// TIA Portal V19 export
VAR_GLOBAL   // PLC tag table "A03_303"
   A0303_Spalla_Ax_Testa_Posizionamento_Ls_Minimo AT %I355.7 : Bool;   // 2262SQ1
   A0303_Spalla_Ax_Testa_Posizionamento_Ls_Massimo AT %I356.0 : Bool;   // 2262SQ2
   A0303_Spintore_Testa_Verticale_Ls_Rest AT %I356.1 : Bool;   // 2270SQ1
   A0303_Spintore_Testa_Verticale_Ls_Work AT %I356.2 : Bool;   // 2270SQ2
   A0303_Spintore_Testa_Orizzontale_Ls_Rest AT %I356.3 : Bool;   // 2270SQ3
   A0303_Spintore_Testa_Orizzontale_Ls_Work AT %I356.4 : Bool;   // 2270SQ4
   A0303_Spintore_Testa_Verticale_V_Rest AT %Q362.2 : Bool;   // 2270YV1
   A0303_Spintore_Testa_Verticale_V_Work AT %Q362.3 : Bool;   // 2270YV2
   A0303_Spintore_Testa_Orizzontale_V_Rest AT %Q362.4 : Bool;   // 2270YV3
   A0303_Spintore_Testa_Orizzontale_V_Work AT %Q362.5 : Bool;   // 2270YV4
   A0303_ControlloPezzo_Testa_Phc_InPosizione AT %I356.5 : Bool;   // 2271BF1
   A0303_ControlloPezzo_Testa_Phc_MassimaPosizione AT %I356.6 : Bool;   // 2271BF2
   A0303_SostegnoStrato_Testa_Verticale_Ls_Alto AT %I356.7 : Bool;   // 2274SQ1
   A0303_SostegnoStrato_Testa_Verticale_Ls_Basso AT %I357.0 : Bool;   // 2274SQ2
   A0303_SostegnoStrato_Testa_Verticale_V_Alto AT %Q362.6 : Bool;   // 2274YV1
   A0303_SostegnoStrato_Testa_Verticale_V_Basso AT %Q362.7 : Bool;   // 2274YV2
   A0303_Spalla_Ax_Coda_Posizionamento_Ls_Minimo AT %I305.7 : Bool;   // 2282SQ1
   A0303_Spalla_Ax_Coda_Posizionamento_Ls_Massimo AT %I306.0 : Bool;   // 2282SQ2
   A0303_Spintore_Coda_Verticale_Ls_Rest AT %I306.1 : Bool;   // 2300SQ1
   A0303_Spintore_Coda_Verticale_Ls_Work AT %I306.2 : Bool;   // 2300SQ2
   A0303_Spintore_Coda_Orizzontale_Ls_Rest AT %I306.3 : Bool;   // 2300SQ3
   A0303_Spintore_Coda_Orizzontale_Ls_Work AT %I306.4 : Bool;   // 2300SQ4
   A0303_Spintore_Coda_Verticale_V_Rest AT %Q311.6 : Bool;   // 2300YV1
   A0303_Spintore_Coda_Verticale_V_Work AT %Q311.7 : Bool;   // 2300YV2
   A0303_Spintore_Coda_Orizzontale_V_Rest AT %Q312.0 : Bool;   // 2300YV3
   A0303_Spintore_Coda_Orizzontale_V_Work AT %Q312.1 : Bool;   // 2300YV4
   A0303_ControlloPezzo_Coda_Phc_InPosizione AT %I306.5 : Bool;   // 2301BF1
   A0303_ControlloPezzo_Coda_Phc_MassimaPosizione AT %I306.6 : Bool;   // 2301BF2
   A0303_SostegnoStrato_Coda_Verticale_Ls_Alto AT %I306.7 : Bool;   // 2304SQ1
   A0303_SostegnoStrato_Coda_Verticale_Ls_Basso AT %I307.0 : Bool;   // 2304SQ2
   A0303_SostegnoStrato_Coda_Verticale_V_Alto AT %Q312.2 : Bool;   // 2304YV1
   A0303_SostegnoStrato_Coda_Verticale_V_Basso AT %Q312.3 : Bool;   // 2304YV2
   A0303_Traslazione_Strato_Ax_Orizzontale_Testa_Ls_Minimo AT %I357.1 : Bool;   // 2312SQ1
   A0303_Traslazione_Strato_Ax_Orizzontale_Testa_Ls_Massimo AT %I357.2 : Bool;   // 2312SQ2
   "A0303_Manipolatore_Strato_Testa_Sostegno_''L''_Ls_Rest" AT %I357.3 : Bool;   // 2320SQ1
   "A0303_Manipolatore_Strato_Testa_Sostegno_''L''_Ls_Work" AT %I357.4 : Bool;   // 2320SQ2
   A0303_Manipolatore_Strato_Testa_Pareggiatore_Ls_Rest AT %I357.5 : Bool;   // 2320SQ3
   A0303_Manipolatore_Strato_Testa_Pareggiatore_Ls_Work AT %I357.6 : Bool;   // 2320SQ4
   "A0303_Manipolatore_Strato_Testa_Sostegno_''L''_V_Rest" AT %Q363.0 : Bool;   // 2320YV1
   "A0303_Manipolatore_Strato_Testa_Sostegno_''L''_V_Work" AT %Q363.1 : Bool;   // 2320YV2
   A0303_Manipolatore_Strato_Testa_Pareggiatore_V_Rest AT %Q363.2 : Bool;   // 2320YV3
   A0303_Manipolatore_Strato_Testa_Pareggiatore_V_Work AT %Q363.3 : Bool;   // 2320YV4
   A0303_Traslazione_Strato_Ax_Orizzontale_Coda_Ls_Minimo AT %I307.1 : Bool;   // 2332SQ1
   A0303_Traslazione_Strato_Ax_Orizzontale_Coda_Ls_Massimo AT %I307.2 : Bool;   // 2332SQ2
   "A0303_Manipolatore_Strato_Coda_Sostegno_''L''_Ls_Rest" AT %I307.3 : Bool;   // 2340SQ1
   "A0303_Manipolatore_Strato_Coda_Sostegno_''L''_Ls_Work" AT %I307.4 : Bool;   // 2340SQ2
   A0303_Manipolatore_Strato_Coda_Pareggiatore_Ls_Rest AT %I307.5 : Bool;   // 2340SQ3
   A0303_Manipolatore_Strato_Coda_Pareggiatore_Ls_Work AT %I307.6 : Bool;   // 2340SQ4
   "A0303_Manipolatore_Strato_Coda_Sostegno_''L''_V_Rest" AT %Q312.4 : Bool;   // 2340YV1
   "A0303_Manipolatore_Strato_Coda_Sostegno_''L''_V_Work" AT %Q312.5 : Bool;   // 2340YV2
   A0303_Manipolatore_Strato_Coda_Pareggiatore_V_Rest AT %Q312.6 : Bool;   // 2340YV3
   A0303_Manipolatore_Strato_Coda_Pareggiatore_V_Work AT %Q312.7 : Bool;   // 2340YV4
   A0303_Posizione_Y_Ax_Testa_Ls_Minimo AT %I357.7 : Bool;   // 2352SQ1
   A0303_Posizione_Y_Ax_Testa_Ls_Massimo AT %I358.0 : Bool;   // 2352SQ2
   A0303_Pistoni_Posizione_1_Paletti_Sostegno_Testa_Ls_Rest AT %I358.1 : Bool;   // 2360SQ1
   A0303_Pistoni_Posizione_1_Paletti_Sostegno_Testa_Ls_Work AT %I358.2 : Bool;   // 2360SQ2
   A0303_Pistoni_Posizione_2_Paletti_Sostegno_Testa_Ls_Rest AT %I358.3 : Bool;   // 2360SQ3 (Libero)
   A0303_Pistoni_Posizione_2_Paletti_Sostegno_Testa_Ls_Work AT %I358.4 : Bool;   // 2360SQ4
   A0303_Pistoni_Posizione_1_Paletti_Sostegno_Testa_V_Rest AT %Q363.4 : Bool;   // 2360YV1
   A0303_Pistoni_Posizione_1_Paletti_Sostegno_Testa_V_Work AT %Q363.5 : Bool;   // 2360YV2
   A0303_Pistoni_Posizione_2_Paletti_Sostegno_Testa_V_Rest AT %Q363.6 : Bool;   // 2360YV3
   A0303_Pistoni_Posizione_2_Paletti_Sostegno_Testa_V_Work AT %Q363.7 : Bool;   // 2360YV4
   A0303_Posizione_Y_Ax_Coda_Ls_Minimo AT %I307.7 : Bool;   // 2372SQ1
   A0303_Posizione_Y_Ax_Coda_Ls_Massimo AT %I308.0 : Bool;   // 2372SQ2
   A0303_Pistoni_Posizione_1_Paletti_Sostegno_Coda_Ls_Rest AT %I308.1 : Bool;   // 2380SQ1
   A0303_Pistoni_Posizione_1_Paletti_Sostegno_Coda_Ls_Work AT %I308.2 : Bool;   // 2380SQ2
   A0303_Pistoni_Posizione_2_Paletti_Sostegno_Coda_Ls_Rest AT %I308.3 : Bool;   // 2380SQ3 (Libero)
   A0303_Pistoni_Posizione_2_Paletti_Sostegno_Coda_Ls_Work AT %I308.4 : Bool;   // 2380SQ4
   A0303_Pistoni_Posizione_1_Paletti_Sostegno_Coda_V_Rest AT %Q313.0 : Bool;   // 2380YV1
   A0303_Pistoni_Posizione_1_Paletti_Sostegno_Coda_V_Work AT %Q313.1 : Bool;   // 2380YV2
   A0303_Pistoni_Posizione_2_Paletti_Sostegno_Coda_V_Rest AT %Q313.2 : Bool;   // 2380YV3
   A0303_Pistoni_Posizione_2_Paletti_Sostegno_Coda_V_Work AT %Q313.3 : Bool;   // 2380YV4
   A0303_Sollevamento_Pacco_Ax_Testa_Ls_Minimo AT %I358.5 : Bool;   // 2392SQ1
   A0303_Sollevamento_Pacco_Ax_Testa_Ls_Massimo AT %I358.6 : Bool;   // 2392SQ2
   A0303_Sollevamento_Pacco_Ax_Coda_Ls_Minimo AT %I308.5 : Bool;   // 2402SQ1
   A0303_Sollevamento_Pacco_Ax_Coda_Ls_Massimo AT %I308.6 : Bool;   // 2402SQ2
   A0303_AI_Manipolatore_Testa_Strato_Phc_Depositato AT %IW942 : Int;   // 552A1 - 2321BF1
   A0303_AI_Manipolatore_Coda_Strato_Phc_Depositato AT %IW938 : Int;   // 533A1 - 2341BF1
END_VAR
